Staubli VAL3: WAGO750_631.pjx

--- WAGO750_631.pjx ---
Parameters version=s7.3 stackSize=5000 millimeterUnit=true
Program file=_DetectIOEdge.pgx
Program file=create.pgx
Program file=enableLatch.pgx
Program file=encoder.pgx
Program file=getResolution.pgx
Program file=getStatus.pgx
Program file=getValue.pgx
Program file=init.pgx
Program file=isLatched.pgx
Program file=kill.pgx
Program file=reset.pgx
Program file=resetLatch.pgx
Program file=setResolution.pgx
Program file=start.pgx
Program file=stop.pgx
Data file=WAGO750_631.dtx

--- WAGO750_631.dtx ---
public aio aiEncCurrentPos = {link=ApplicomIO-1\ENCODER-BLOCKC\%IW1}
aio aiEncLatchedPos = {link=ApplicomIO-1\ENCODER-BLOCKC\%IW4}
aio aoEncResolution
aio aoPresetPos = {link=ApplicomIO-1\ENCODER-BLOCKC\%QW1}
public bool bLatchEnabled
bool bMemoLatchState
bool bMemoOvf
bool bMemoUdf
bool bPartLatched
bool bReset
dio diEncLatched = {link=ApplicomIO-1\ENCODER-BLOCKC\%I1}
dio diOverFlow = {link=ApplicomIO-1\ENCODER-BLOCKC\%I4}
dio diPresetACK = {link=ApplicomIO-1\ENCODER-BLOCKC\%I2}
dio diUnderFlow = {link=ApplicomIO-1\ENCODER-BLOCKC\%I3}
dio doEnableLatch = {link=ApplicomIO-1\ENCODER-BLOCKC\%Q1}
dio doEnablePreset = {link=ApplicomIO-1\ENCODER-BLOCKC\%Q2}
num nEncLatchedVal = 1
num nEncResolution = 1024
num nEncValue = 1
public num nLatchPeriod = 1
public num nMAXCOUNT
public num nMINCOUNT
num nPresetPos = 1
string sEncNum
string sTASK = "encoder"
